(* PLC project liner_cyclic.project, CODESYS CODESYS V3.5 SP17 Patch 3 *)
(* stored: creationDateTime 1970-01-01T00:00:00, modificationDateTime 1970-01-01T00:00:00 *)

{attribute 'qualified_only'}
{attribute 'strict'}
TYPE State : (INIT := 0, RUNNING := 1, COMPLETE := 2);
END_TYPE
